(* IEC 61131-3 sources: Std_PalletMover/Class/Per_Hal_Bms_MasterVolt, 1 file *)

(* ---- Per_Hal_Bms_MasterVolt.st ---- *)
(*!
<Class
	Name               = "Per_Hal_Bms_MasterVolt"
	Revision           = "0.0"
	RealtimeTask       = "false"
	CyclicTask         = "false"
	BackgroundTask     = "false"
	Sigmatek           = "false"
	OSInterface        = "false"
	HighPriority       = "false"
	Automatic          = "false"
	UpdateMode         = "Prescan"
	SharedCommandTable = "true"
	Objectsize         = "(750,180)">
	<Channels>
		<Server Name="BmsInterface" Class="HalBmsMastervoltinterface" Visualized="false" Initialize="false" WriteProtected="true" Retentive="false"/>
		<Server Name="ClassSvr" Visualized="false" Initialize="false" WriteProtected="true" Retentive="false"/>
		<Client Name="Driver" Required="false" Internal="false"/>
		<Client Name="HAL_BMS_MasterVolt" Required="true" Internal="true"/>
		<Client Name="ObjHalBmsMastervoltinterface" Required="true" Internal="true"/>
		<Client Name="op_LogData" Required="false" Internal="false" Comment="Output for logging data to SF_Logger"/>
		<Client Name="p_NextObject" Required="false" Internal="false" Comment="Pointer to next object in linked list"/>
	</Channels>
	<Network Name="Per_Hal_Bms_MasterVolt">
		<!-- List of Components in this network -->
		<Components>
			<Object
				Name       = "HAL_BMS_MasterVolt"
				Class      = "HAL_BMS_MasterVolt"
				Position   = "(454,90)"
				Visualized = "true"
				CyclicTime = "100 ms">
				<Channels>
					<Server Name="BatteryAlarms"/>
					<Server Name="BatteryCharging"/>
					<Server Name="BatteryCurrent"/>
					<Server Name="BatteryTemperature"/>
					<Server Name="BatteryVirtualStateOfCharge"/>
					<Server Name="BatteryVoltage"/>
					<Server Name="ClassSvr"/>
					<Server Name="EnergyDraw"/>
					<Server Name="HMIAdditionalIcon"/>
					<Server Name="HMIIconState"/>
					<Server Name="LowBatteryLimit" Value="40"/>
					<Server Name="NMT"/>
					<Server Name="StateOfCharge"/>
					<Client Name="cNode" Value="32"/>
					<Client Name="Driver"/>
				</Channels>
			</Object>
			<Object
				Name       = "ObjHalBmsMastervoltinterface"
				Class      = "HalBmsMastervoltinterface"
				Position   = "(450,1140)"
				Visualized = "false">
				<Channels>
					<Server Name="ClassSvr"/>
					<Client Name="ToBmsMastervolt"/>
				</Channels>
			</Object>
		</Components>
		<Comments>
		</Comments>
		<!-- List of Connections in this network -->
		<Connections>
			<Connection Source="this.HAL_BMS_MasterVolt" Destination="HAL_BMS_MasterVolt.ClassSvr"/>
			<Connection Source="this.ObjHalBmsMastervoltinterface" Destination="ObjHalBmsMastervoltinterface.ClassSvr"/>
			<Connection Source="HAL_BMS_MasterVolt.Driver" Destination="this.Driver" Vertices="(454,180),(38,210),"/>
			<Connection Source="this.BmsInterface" Destination="ObjHalBmsMastervoltinterface.ClassSvr" Vertices="(1482,270),(1306,1230),"/>
			<Connection Source="ObjHalBmsMastervoltinterface.ToBmsMastervolt" Destination="HAL_BMS_MasterVolt.ClassSvr" Vertices="(450,1230),(1310,180),"/>
		</Connections>
		<!-- Headerfiles -->
		<Options>
		</Options>
	</Network>
</Class>
*)
Per_Hal_Bms_MasterVolt : CLASS
  //Servers:
	ClassSvr 	: SvrChCmd_DINT;
	BmsInterface 	: SvrChCmd_DINT;
  //Clients:
	HAL_BMS_MasterVolt 	: CltChCmd_HAL_BMS_MasterVolt;
	Driver 	: CltChCmd_CanDriverBase;
	op_LogData 	: CltCh_gpt_LogData;
	p_NextObject 	: CltChCmd_LinkedObjectBase;
	ObjHalBmsMastervoltinterface 	: CltChCmd_HalBmsMastervoltinterface;
  //Variables:
  //Functions:

	FUNCTION VIRTUAL GLOBAL BmsInterface::Read
		VAR_OUTPUT
			output (EAX) 	: DINT;
		END_VAR;
  //Tables:
	FUNCTION @STD
		VAR_OUTPUT
			ret_code	: CONFSTATES;
		END_VAR;
	FUNCTION GLOBAL TAB @CT_;
END_CLASS;

#pragma using HAL_BMS_MasterVolt
#pragma using HalBmsMastervoltinterface
#pragma usingLtd CanDriverBase
#pragma usingLtd LinkedObjectBase

FUNCTION VIRTUAL GLOBAL Per_Hal_Bms_MasterVolt::BmsInterface::Read
	VAR_OUTPUT
		output (EAX) 	: DINT;
	END_VAR

	BmsInterface := ObjHalBmsMastervoltinterface.ClassSvr.Read();
	output := BmsInterface;

END_FUNCTION
